FUNCTION_BLOCK AxesFeedback EXTENDS SM_AxesFeedback
VAR_INPUT
END_VAR
VAR_OUTPUT
END_VAR
VAR
END_VAR

SUPER^();

END_FUNCTION_BLOCK

(* stored: Version 1.1.0.1, ProductVersion 3.1.4019.2
   POU AxesFeedback: Id {5f29066f-bccb-4802-b6c3-b32cfba28831}, SpecialFunc None *)
